Staubli VAL3: AxisTest.pgx

public program AxisTest()
begin
  dDio["O1_bFollowOn"]=true
  delay(0.5)
  dDio["O1_bFollowOn"]=false
  delay(0.5)
  dDio["O1_bFollowOn"]=true
  delay(0.5)
  dDio["O1_bFollowOn"]=false
  delay(0.5)


end
